// TIA Portal V20 export
DATA_BLOCK "TestIo_DB"   // DB306
// stored: AutoNumber false, InstanceOfName TestIo, InstanceOfType FB
"TestIo"
BEGIN
END_DATA_BLOCK
